(* IEC 61131-3 sources: eCockpitGit/test_project/src/%F%00 Library/%F%Common Functions/%F%Math/%F%Average, 5 files *)

(* ---- %POU%FU_diAverage.st ---- *)
//This calculates the average of a stream of numbers
//Must be used like this average := FU_iAvarage(lastAverage:=average,newValue:=value,count:=count);
//Count starts at 1
// |**Version**|**Author**| **Date** |**Changes**
// | 1         | NSN      | 12-01-21 | creation
FUNCTION FU_diAverage : DINT
VAR_INPUT
	lastAverage		:DINT;
	newValue		:DINT;
	count			:BYTE;
END_VAR
(*%!%__DELIMITER__%!%*)
FU_diAverage := (lastAverage +  (newValue - lastAverage) / count + 1) - 1;

(* ---- %POU%FU_diAverageOfTwo.st ---- *)
//This function calculates The average of the two inputs
// +-----------+----------+----------+-----------------------------------------------------------------------------------------------------------------------+
// |**Version**|**Author**| **Date** |**Changes**                                                                                                            |
// +-----------+----------+----------+-----------------------------------------------------------------------------------------------------------------------+
// | 1         | NSN      | 11-12-18 | Creation                                                                                                              |
// +-----------+----------+----------+-----------------------------------------------------------------------------------------------------------------------+
FUNCTION FU_diAverageOfTwo : DINT
VAR_INPUT
	iA			:DINT;	//Value A
	iB			:DINT;	//Value B
END_VAR
(*%!%__DELIMITER__%!%*)
FU_diAverageOfTwo := (iA+iB)/2;

(* ---- %POU%FU_iAverage.st ---- *)
//This calculates the average of a stream of numbers
//Must be used like this average := FU_iAvarage(lastAverage:=average,newValue:=value,count:=count);
//Count starts at 1
// |**Version**|**Author**| **Date** |**Changes**
// | 1         | NSN      | 12-01-21 | creation
FUNCTION FU_iAverage : INT
VAR_INPUT
	lastAverage		:INT;
	newValue		:INT;
	count			:BYTE;
END_VAR
(*%!%__DELIMITER__%!%*)
FU_iAverage := (lastAverage + (newValue - lastAverage) / count + 1) - 1;

(* ---- %POU%FU_iAverageOfTwo.st ---- *)
//This function calculates The average of the two inputs
// +-----------+----------+----------+-----------------------------------------------------------------------------------------------------------------------+
// |**Version**|**Author**| **Date** |**Changes**                                                                                                            |
// +-----------+----------+----------+-----------------------------------------------------------------------------------------------------------------------+
// | 1         | NSN      | 20-09-18 | Updated to new format                                                                                                 |
// +-----------+----------+----------+-----------------------------------------------------------------------------------------------------------------------+
FUNCTION FU_iAverageOfTwo : INT
VAR_INPUT
	iA			:INT;	//Value A
	iB			:INT;	//Value B
END_VAR
(*%!%__DELIMITER__%!%*)
FU_iAverageOfTwo := (iA+iB)/2;

(* ---- %POU%FU_rAverage.st ---- *)
//This calculates the average of a stream of numbers
//Must be used like this average := FU_iAvarage(lastAverage:=average,newValue:=value,count:=count);
//Count starts at 1
// |**Version**|**Author**| **Date** |**Changes**
// | 1         | NSN      | 12-01-21 | creation
FUNCTION FU_rAverage : REAL
VAR_INPUT
	lastAverage		:REAL;
	newValue		:REAL;
	count			:BYTE;
END_VAR
(*%!%__DELIMITER__%!%*)
FU_rAverage := (lastAverage +  (newValue - lastAverage) / count + 1) - 1;
